FUNCTION_BLOCK TEvent_AssertionFailed EXTENDS TEventBase IMPLEMENTS IEvent
VAR
    Message : T_MaxString;
    Handler : IEventHandler_OnAssertionFailed;
END_VAR

METHOD  CallHandler
VAR_INPUT
    HandlerBase : IEventHandlerBase;
    EventArgs   : IStreamReader;
END_VAR
IF __QUERYINTERFACE(HandlerBase,Handler) THEN
    Message := EventArgs.Read_STRING();
    Handler.OnAssertionFailed(EventArgs);
END_IF
END_METHOD

METHOD  IsHandlerSupported : BOOL
VAR_INPUT
    HandlerBase : IEventHandlerBase;
END_VAR
IF __QUERYINTERFACE(HandlerBase,Handler) THEN
    IsHandlerSupported := TRUE;
END_IF
END_METHOD

END_FUNCTION_BLOCK

(* stored: Version 1.1.0.1, ProductVersion 3.1.4024.3
   POU TEvent_AssertionFailed: Id {c96590be-9346-4ddc-943b-792d0d6d2694}, SpecialFunc None
   Method CallHandler: Id {a2f509c9-1ae1-4969-9c62-873357bc1858}
   Method IsHandlerSupported: Id {626a8e4e-c8e5-43f4-8c6c-36eeb6e42fa0} *)
